ABB RAPID module: TCPZ_toolBJC.MOD

MODULE TCPZ_toolBJC
	! Points are read in order of declaration.
  ! Please do not change the order of points!

  LOCAL PERS robtarget pTCPZ_Point1:=[[-274.2829,-473.5635,161.5131],[0.380540668964386,0.56345534324646,0.314760655164719,-0.662293434143066],[-2,-2,2,0],[9E+09,9E+09,9E+09,9E+09,9E+09,9E+09]];
	LOCAL PERS robtarget pTCPZ_Point2:=[[-271.6045,-481.7277,242.6312],[0.02209797129035,0.417950481176376,0.658490478992462,-0.625475347042084],[-2,-2,1,0],[9E+09,9E+09,9E+09,9E+09,9E+09,9E+09]];
	LOCAL PERS robtarget pTCPZ_Point3:=[[-346.9195,-479.5418,301.8599],[0.405778437852859,0.80945235490799,0.3222416639328,-0.276208281517029],[-2,-1,0,1],[9E+09,9E+09,9E+09,9E+09,9E+09,9E+09]];
	LOCAL PERS robtarget pTCPZ_Point4:=[[-469.9561,-562.5878,355.5264],[0.328976601362228,0.730729699134827,0.598095893859863,0.00947600230574608],[-2,-2,1,1],[9E+09,9E+09,9E+09,9E+09,9E+09,9E+09]];
	LOCAL PERS robtarget pTCPZ_ElongZ:=[[-331.187,-519.6253,343.3361],[0.21037483215332,0.746861457824707,0.543452382087708,-0.320312142372131],[-2,-2,1,1],[9E+09,9E+09,9E+09,9E+09,9E+09,9E+09]];


! Tool
TASK PERS tooldata toolBJC:=[TRUE,[[7.62994,4.36555,211.035],[0.819285,0.523964,-0.19619,-0.125471]],[-1,[0,0,0],[1,0,0,0],0,0,0]];

ENDMODULE
